PROGRAM MAIN
VAR
  bInit                     : BOOL;         // shall be checked by controlling entity, before using Ctrl/State structs
  eInit                     : E_PROGRESS;   // shall be checked by controlling entity, before using Ctrl/State structs

  nAxis,
  nAxisInit                 : UINT;

  stMsg                     : ST_Message;

  bWriteTimerActive         : Bool;         // you decide whether to use timed logging into file or not
  tWriteLog                 : TIME := T#10S;
  tonWriteLog               : Tc2_Standard.TON;
END_VAR


(*
//-----------------------------------------------------------------------------------------------------------------
//-----------------------------------------------------------------------------------------------------------------
// react to operation modes (how to do it in an easy self documenting way)
//-----------------------------------------------------------------------------------------------------------------
//-----------------------------------------------------------------------------------------------------------------
CASE (GVL_AXIS.State[i].eState MOD E_PROGRESS.PROGRESS_DONE)
OF
  E_AXIS_STATE.AXIS_INIT:
    ;// do something after success  

  E_AXIS_STATE.AXIS_MOVE_POS::
    ;// do something after success
ELSE
  CASE (GVL_AXIS.State[i].eState MOD E_PROGRESS.PROGRESS_ERROR)
  OF
    E_AXIS_STATE.AXIS_INIT:
      ;// do something after success  
  
    E_AXIS_STATE.AXIS_MOVE_POS::
      ;// do something after success
  ELSE
    ;// down the rabbit hole you go from here
  END_CASE
END_CASE
*)



//-----------------------------------------------------------------------------------------------------------------
// Local time; used for timestamps
//-----------------------------------------------------------------------------------------------------------------
GVL_MSG.fbLocalTime(
                    sLocalTime                => GVL_MSG.sLocalTime, 
                    dtLocalTime               => GVL_MSG.dtLocalTime);
//-----------------------------------------------------------------------------------------------------------------
//-----------------------------------------------------------------------------------------------------------------
// /assign dataflow
//-----------------------------------------------------------------------------------------------------------------
FOR nAxis := 1 TO PLC_CONSTANT.MAX_AXIS
DO
  GVL_AXIS.Control[nAxis].AxisIndex           := nAxis;

  GVL_AXIS.Control[nAxis].AxisCtrl            := ADR(GVL_AXIS.Ctrl);          // command
  GVL_AXIS.Control[nAxis].AxisState           := ADR(GVL_AXIS.State);         // state + result of command

  GVL_AXIS.Control[nAxis].Axes                REF=   GVL_AXIS.AxisRef;        // All for one; coupling requires access across all axes

  GVL_AXIS.Control[nAxis].AxisInfo            := ADR(GVL_AXIS.Info);          // axis information: act/set values and bits from axis
  GVL_AXIS.Control[nAxis].AxisData            := ADR(GVL_AXIS.Data);          // position and dynamic constraints for movement
  GVL_AXIS.Control[nAxis].AxisGearInParameter := ADR(GVL_AXIS.GearInParameter);

  GVL_AXIS.Control[nAxis].WriteNcParameter    := ADR(GVL_AXIS.NcParameterWrt);
  GVL_AXIS.Control[nAxis].ReadNcParameter     := ADR(GVL_AXIS.NcParameterRd);

  GVL_AXIS.Control[nAxis].HomingParameter     := ADR(GVL_AXIS.HomeParameter);
  GVL_AXIS.Control[nAxis].MotionOptions       := ADR(GVL_AXIS.MotionOptions);

  GVL_AXIS.ItfMcAxis[nAxis]                   := GVL_AXIS.Control[nAxis]; 
END_FOR
//-----------------------------------------------------------------------------------------------------------------
// assign dataflow/
//-----------------------------------------------------------------------------------------------------------------
//-----------------------------------------------------------------------------------------------------------------
// /INIT
// - successful init is required for other optional members to start
//-----------------------------------------------------------------------------------------------------------------
IF NOT bInit
THEN
  CASE eInit
  OF
    E_PROGRESS.PROGRESS_INVALID,
    E_PROGRESS.PROGRESS_DONE:
      FOR nAxis := 1 TO PLC_CONSTANT.MAX_AXIS
      DO
        GVL_AXIS.Control[nAxis].MessageLevel  := GVL_MSG.MessageLevelAxisPtp;
      END_FOR
      nAxisInit                               := 1;
      eInit                                   := E_PROGRESS.PROGRESS_INIT;


    E_PROGRESS.PROGRESS_INIT:
      stMsg.eType                             := E_MessageType.eMessageVerbose;
      stMsg.eDevice                           := e_Device.General;
      stMsg.eSubdevice                        := e_SubDevice.AxisStartUp;
      stMsg.iErrorNumber                      := nAxisInit;

      stMsg.sText                             := concat('MAIN.eInit: ', TO_STRING(eInit));

      IF (GVL_MSG.MessageLevelAxisPtp = E_MessageType.eMessageVerbose)
      THEN
        f_MessageSet(stMsg);
      END_IF

      GVL_AXIS.Ctrl[nAxisInit].eCmd           := E_AXIS_CTRL.AXIS_NULL;
      eInit                                   := E_PROGRESS.PROGRESS_BUSY;


    E_PROGRESS.PROGRESS_BUSY:
      GVL_AXIS.Ctrl[nAxisInit].eCmd          := E_AXIS_CTRL.AXIS_INIT;

      IF    (GVL_AXIS.State[nAxisInit].eState = E_AXIS_STATE.AXIS_INIT + E_PROGRESS.PROGRESS_ERROR)
      THEN
        eInit                                 := E_PROGRESS.PROGRESS_ERROR;

        stMsg.eType                           := E_MessageType.eMessageError;
        stMsg.eDevice                         := e_Device.General;
        stMsg.eSubdevice                      := e_SubDevice.AxisStartUp;
        stMsg.iErrorNumber                    := GVL_AXIS.Control[nAxisInit].ErrorId;

        stMsg.sText                           := concat('MAIN.eInit ERROR at Index: ', TO_STRING(nAxisInit));
        f_MessageSet(stMsg);

      ELSIF (GVL_AXIS.State[nAxisInit].eState = E_AXIS_STATE.AXIS_INIT + E_PROGRESS.PROGRESS_DONE)
      THEN
        eInit                                 := E_PROGRESS.PROGRESS_CHECK;
      END_IF


    E_PROGRESS.PROGRESS_CHECK:
      IF NOT (nAxisInit > PLC_CONSTANT.MAX_AXIS-1)
      THEN
        nAxisInit                             := nAxisInit + 1;
        eInit                                 := E_PROGRESS.PROGRESS_INIT;

      ELSE
        bInit                                 := TRUE;
        eInit                                 := E_PROGRESS.PROGRESS_DONE;

        stMsg.eType                           := E_MessageType.eMessageInfo;
        stMsg.eDevice                         := e_Device.General;
        stMsg.eSubdevice                      := e_SubDevice.AxisStartUp;
        stMsg.iErrorNumber                    := MAX_AXIS;

        stMsg.sText                           := concat('MAIN.eInit: ', TO_STRING(eInit));
        f_MessageSet(stMsg);
      END_IF
  END_CASE
END_IF
//-----------------------------------------------------------------------------------------------------------------
// INIT
//-----------------------------------------------------------------------------------------------------------------
//-----------------------------------------------------------------------------------------------------------------
// /cyclic
//-----------------------------------------------------------------------------------------------------------------
IF (eInit <> E_PROGRESS.PROGRESS_ERROR)
THEN
  FOR nAxis := 1 TO PLC_CONSTANT.MAX_AXIS
  DO
      GVL_AXIS.Control[nAxis]();
  END_FOR
END_IF
//-----------------------------------------------------------------------------------------------------------------
// cyclic/
//-----------------------------------------------------------------------------------------------------------------


//-----------------------------------------------------------------------------------------------------------------
// /logging
//-----------------------------------------------------------------------------------------------------------------
tonWriteLog(IN:= TRUE, PT := tWriteLog);

IF (tonWriteLog.Q)
THEN
  MessageData.bWriteFile      := bWriteTimerActive; // you have to decide whether to use timed write or not
  tonWriteLog(IN:= FALSE);
END_IF

//-----------------------------------------------------------------------------------------------------------------
// write message list to file
//-----------------------------------------------------------------------------------------------------------------
MessageData(pList			        := ADR(GVL_MSG.Messages),
			      pLocalTime        := ADR(GVL_MSG.dtLocalTime), 
			      bBusy=> );

// clear write trigger
IF MessageData.bWriteFile AND
   MessageData.bBusy
THEN
  MessageData.bWriteFile      := FALSE;
END_IF
//-----------------------------------------------------------------------------------------------------------------
// logging/
//-----------------------------------------------------------------------------------------------------------------

END_PROGRAM

(* stored: Version 1.1.0.1, ProductVersion 3.1.4026.13
   POU MAIN: Id {b9c2507d-2926-4719-8f82-549e0347748a}, SpecialFunc None *)
